ABB RobotStudio station: Lab5_RSSolution.rspag

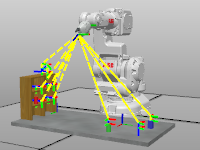
--- station ---
Station Lab5_RSSolution (saved by RobotStudio 20.4.9280.0)
Controller Lab5Controller
  mechanical unit ROB_1: IRB140_6_81_C_03, 6 joints, base frame (0, 0, 0) mm
Layout (positions relative to the parent item):
  - IRB140_6_81_C_03 [mechanism, from Robots\IRB140_6_81_C_G_03.rslib] at (0, 0, 0) mm; joint values [0, 0, 0, 0, 0.5236, 0] (rad or m)
  - HorizontalPlaneBoard [part]
  - WoodenRack [part]
  - PrismPiece [part] at (380, 400, 25) mm
  - CylinderPiece [part] at (580, 200, 25) mm, rotated rx 0 ry 0 rz -90 deg
  - HexagonalPrismPiece [part] at (502.54, -420.19, 127.78) mm, rotated rx 0 ry 0 rz -1.03 deg
  - Smart_Gripper_Servo_Fingers [mechanism, from Libraries\Smart_Gripper_Servo_Fingers.rslib] at (506.29, 0, 679.5) mm, rotated rx 180 ry 60 rz 180 deg; joint values [0.025] (rad or m)
  - PickAndPlaceLogic [smart component]
      signals: DI ActivateGripper, DI ReleaseGripper, DO PieceTaken
      connections:
        PickAndPlaceLogic.ActivateGripper -> Attacher.Execute
        PickAndPlaceLogic.ReleaseGripper -> Detacher.Execute
    - Attacher [smart component, from Components\Attacher.rslib]
        properties: Parent=Smart_Gripper_Servo_Fingers; Flange=0; Child=HexagonalPrismPiece; Mount=false; Offset=[0 0 0]; Orientation=[0 0 0]
    - Detacher [smart component, from Components\Detacher.rslib]
        properties: Child=HexagonalPrismPiece; KeepPosition=true
Attachment: Smart_Gripper_Servo_Fingers is attached to IRB140_6_81_C_03 / Link6
Station logic (signal -> signal, property => property):
  PickAndPlaceLogic.PieceTaken -> Lab5Controller.DI_01
  Lab5Controller.DO_02 -> PickAndPlaceLogic.ReleaseGripper
  Lab5Controller.DO_01 -> PickAndPlaceLogic.ActivateGripper

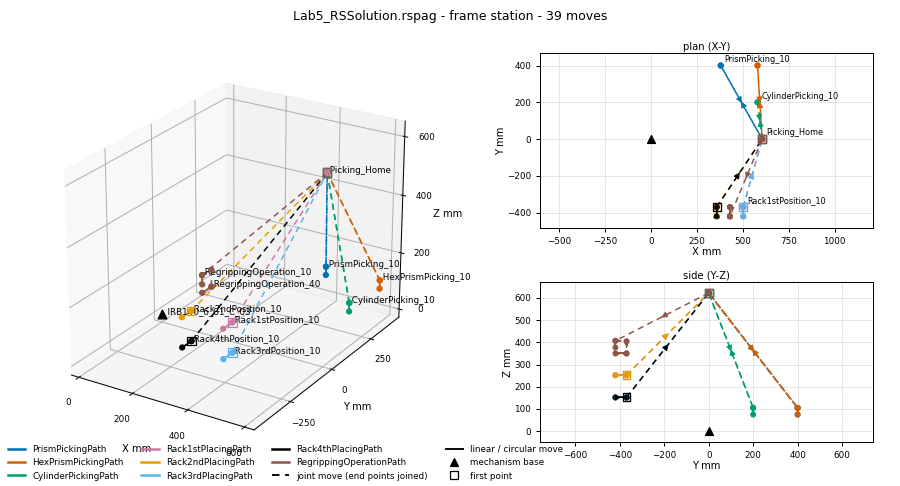
[picture p0: tool path of Lab5_RSSolution.rspag in frame station, 39 of 39 moves have a stored position in this frame; points joined in program order, loops and branches not executed]
--- Backups/Lab5Controller/RAPID/TASK1/PROGMOD/Module1.mod ---
MODULE Module1
        PERS tooldata Servo:=[TRUE,[[0,0,114.2],[1,0,0,0]],[0.215,[8.7,12.3,49.2],[1,0,0,0],0.00021,0.00024,0.00009]];
    TASK PERS wobjdata RackWorkObject:=[FALSE,TRUE,"",[[280,-400,25],[0.707107,0,0,-0.707107]],[[0,0,0],[1,0,0,0]]];
    TASK PERS wobjdata PiecesWorkObject:=[FALSE,TRUE,"",[[380,200,25],[1,0,0,0]],[[0,0,0],[1,0,0,0]]];
    CONST robtarget Picking_Home:=[[225.191752358,-200,597.4],[0.5,0,0.866025404,0],[0,0,0,0],[9E+09,9E+09,9E+09,9E+09,9E+09,9E+09]];
    CONST robtarget PrismPicking_10:=[[0,200,80],[0,0,1,0],[0,0,0,0],[9E+09,9E+09,9E+09,9E+09,9E+09,9E+09]];
    CONST robtarget PrismPicking_20:=[[0,200,50],[0,0,1,0],[0,0,0,0],[9E+09,9E+09,9E+09,9E+09,9E+09,9E+09]];
    CONST robtarget HexPrismPicking_10:=[[200,200,80],[0,0.258819045,0.965925826,0],[0,0,0,0],[9E+09,9E+09,9E+09,9E+09,9E+09,9E+09]];
    CONST robtarget HexPrismPicking_20:=[[200,200,50],[0,0.258819045,0.965925826,0],[0,0,0,0],[9E+09,9E+09,9E+09,9E+09,9E+09,9E+09]];
    CONST robtarget CylinderPicking_10:=[[200,0,80],[0,0.707106781,0.707106781,0],[0,0,1,0],[9E+09,9E+09,9E+09,9E+09,9E+09,9E+09]];
    CONST robtarget CylinderPicking_20:=[[200,0,50],[0,0.707106781,0.707106781,0],[0,0,0,0],[9E+09,9E+09,9E+09,9E+09,9E+09,9E+09]];
    CONST robtarget Rack1stPosition_10:=[[-30,222.5,227],[0.5,-0.5,0.5,-0.5],[-1,-2,0,0],[9E+09,9E+09,9E+09,9E+09,9E+09,9E+09]];
    CONST robtarget Rack1stPosition_20:=[[20,222.5,227],[0.5,-0.5,0.5,-0.5],[-1,-2,0,0],[9E+09,9E+09,9E+09,9E+09,9E+09,9E+09]];
    CONST robtarget Placing_Home:=[[-400,325.191800236,597.400057165],[0.353553394,-0.612372434,0.612372434,0.353553394],[0,0,0,0],[9E+09,9E+09,9E+09,9E+09,9E+09,9E+09]];
    CONST robtarget Rack2ndPosition_10:=[[-30,77.5,227],[0.5,-0.5,0.5,-0.5],[-1,-2,0,0],[9E+09,9E+09,9E+09,9E+09,9E+09,9E+09]];
    CONST robtarget Rack2ndPosition_20:=[[20,77.5,227],[0.5,-0.5,0.5,-0.5],[-1,-2,0,0],[9E+09,9E+09,9E+09,9E+09,9E+09,9E+09]];
    CONST robtarget Rack3rdPosition_10:=[[-30,222.5,127],[0.5,-0.5,0.5,-0.5],[-1,-2,0,0],[9E+09,9E+09,9E+09,9E+09,9E+09,9E+09]];
    CONST robtarget Rack3rdPosition_20:=[[20,222.5,127],[0.5,-0.5,0.5,-0.5],[-1,-2,0,0],[9E+09,9E+09,9E+09,9E+09,9E+09,9E+09]];
    CONST robtarget Rack4thPosition_10:=[[-30,77.5,127],[0.5,-0.5,0.5,-0.5],[-1,-2,0,0],[9E+09,9E+09,9E+09,9E+09,9E+09,9E+09]];
    CONST robtarget Rack4thPosition_20:=[[20,77.5,127],[0.5,-0.5,0.5,-0.5],[-1,-2,0,0],[9E+09,9E+09,9E+09,9E+09,9E+09,9E+09]];
    CONST robtarget RegrippingOperation_10:=[[20,150,382],[0,-0.707106781,0.707106781,0],[0,0,0,0],[9E+09,9E+09,9E+09,9E+09,9E+09,9E+09]];
    CONST robtarget RegrippingOperation_20:=[[20,150,352],[0,-0.707106781,0.707106781,0],[-1,0,-1,0],[9E+09,9E+09,9E+09,9E+09,9E+09,9E+09]];
    CONST robtarget RegrippingOperation_30:=[[-30,150,380],[0.27059805,-0.653281482,0.653281482,-0.27059805],[-1,-2,0,0],[9E+09,9E+09,9E+09,9E+09,9E+09,9E+09]];
    CONST robtarget RegrippingOperation_40:=[[-30,150,325],[0.5,-0.5,0.5,-0.5],[-1,-2,0,0],[9E+09,9E+09,9E+09,9E+09,9E+09,9E+09]];
    CONST robtarget RegrippingOperation_50:=[[20,150,325],[0.5,-0.5,0.5,-0.5],[-1,-2,0,0],[9E+09,9E+09,9E+09,9E+09,9E+09,9E+09]];


    PROC main()
        WaitDI DI_01, 1;
        HexPrismPickingPath;
        RegrippingOperationPath;
        Rack3rdPlacingPath;
    ENDPROC
    PROC PrismPickingPath()
        MoveJ Picking_Home,v200,z10,Servo\WObj:=PiecesWorkObject;
        MoveJ PrismPicking_10,v200,z10,Servo\WObj:=PiecesWorkObject;
        MoveL PrismPicking_20,v20,z1,Servo\WObj:=PiecesWorkObject;
        MoveL PrismPicking_10,v20,z1,Servo\WObj:=PiecesWorkObject;
        MoveJ Picking_Home,v200,z10,Servo\WObj:=PiecesWorkObject;
    ENDPROC
    PROC HexPrismPickingPath()
        MoveJ Picking_Home,v200,z10,Servo\WObj:=PiecesWorkObject;
        MoveJ HexPrismPicking_10,v200,z10,Servo\WObj:=PiecesWorkObject;
        MoveL HexPrismPicking_20,v20,z1,Servo\WObj:=PiecesWorkObject;
        setDO DO_01, 1;
        WaitTime 1;
        SetDO DO_01, 0;
        MoveL HexPrismPicking_10,v20,z1,Servo\WObj:=PiecesWorkObject;
        MoveJ Picking_Home,v200,z10,Servo\WObj:=PiecesWorkObject;
    ENDPROC
    PROC CylinderPickingPath()
        MoveJ Picking_Home,v200,z10,Servo\WObj:=PiecesWorkObject;
        MoveJ CylinderPicking_10,v200,z10,Servo\WObj:=PiecesWorkObject;
        MoveL CylinderPicking_20,v20,z1,Servo\WObj:=PiecesWorkObject;
        MoveL CylinderPicking_10,v20,z1,Servo\WObj:=PiecesWorkObject;
        MoveJ Picking_Home,v200,z10,Servo\WObj:=PiecesWorkObject;
    ENDPROC
    PROC Rack1stPlacingPath()
        MoveJ Rack1stPosition_10,v200,z10,Servo\WObj:=RackWorkObject;
        MoveL Rack1stPosition_20,v20,z1,Servo\WObj:=RackWorkObject;
        MoveL Rack1stPosition_10,v20,z1,Servo\WObj:=RackWorkObject;
        MoveJ Placing_Home,v200,z10,Servo\WObj:=RackWorkObject;
    ENDPROC
    PROC Rack2ndPlacingPath()
        MoveJ Rack2ndPosition_10,v200,z10,Servo\WObj:=RackWorkObject;
        MoveL Rack2ndPosition_20,v20,z1,Servo\WObj:=RackWorkObject;
        MoveL Rack2ndPosition_10,v20,z1,Servo\WObj:=RackWorkObject;
        MoveJ Placing_Home,v200,z10,Servo\WObj:=RackWorkObject;
    ENDPROC
    PROC Rack3rdPlacingPath()
        MoveJ Rack3rdPosition_10,v200,z10,Servo\WObj:=RackWorkObject;
        MoveL Rack3rdPosition_20,v20,z1,Servo\WObj:=RackWorkObject;
        SetDO DO_02, 1;
        WaitTime 1;
        SetDO DO_02, 0;
        MoveL Rack3rdPosition_10,v20,z1,Servo\WObj:=RackWorkObject;
        MoveJ Placing_Home,v200,z10,Servo\WObj:=RackWorkObject;
    ENDPROC
    PROC Rack4thPlacingPath()
        MoveJ Rack4thPosition_10,v200,z10,Servo\WObj:=RackWorkObject;
        MoveL Rack4thPosition_20,v20,z1,Servo\WObj:=RackWorkObject;
        MoveL Rack4thPosition_10,v20,z1,Servo\WObj:=RackWorkObject;
        MoveJ Placing_Home,v200,z10,Servo\WObj:=RackWorkObject;
    ENDPROC
    PROC RegrippingOperationPath()
        MoveJ Placing_Home,v200,z10,Servo\WObj:=RackWorkObject;
        MoveJ RegrippingOperation_10,v200,z10,Servo\WObj:=RackWorkObject;
        MoveL RegrippingOperation_20,v20,z1,Servo\WObj:=RackWorkObject;
        SetDO DO_02, 1;
        WaitTime 1;
        SetDO DO_02, 0;
        MoveL RegrippingOperation_10,v20,z1,Servo\WObj:=RackWorkObject;
        MoveJ RegrippingOperation_30,v200,z10,Servo\WObj:=RackWorkObject;
        MoveJ RegrippingOperation_40,v200,z10,Servo\WObj:=RackWorkObject;
        MoveL RegrippingOperation_50,v20,z1,Servo\WObj:=RackWorkObject;
        SetDO DO_01, 1;
        WaitTime 1;
        SetDO DO_01, 0;
        MoveL RegrippingOperation_40,v20,z1,Servo\WObj:=RackWorkObject;
    ENDPROC
ENDMODULE

--- Backups/Lab5Controller/RAPID/TASK1/SYSMOD/LINKEDM.sys ---
%%%
  VERSION:1
  LANGUAGE:ENGLISH
%%%

MODULE LINKEDM (SYSMODULE)

! FOLLOWER
!     Name of electronically linked follower axis used by operator at teach pendent.
      PERS string l_f_axis_name{5}       :=  ["",  "", "", "", ""];

!     Name of the mechanical unit for follower axis.
      PERS string l_f_mecunt_n{5}  :=  ["", "", "", "", ""];

!     Linked follower axis number in the mechanical unit (first axis in mech. unit is number 1).
      PERS num l_f_axis_no{5}      :=  [0,          0,   0,  0,  0];

! MASTER
!     Name of the mechanical unit for linked master axis.
      PERS string l_m_mecunt_n{5} :=  ["", "", "", "", ""];

!     Linked master axis number in the mechanical unit (first axis in mech. unit is number 1).
!     See axis number table in documentation for different master mechanical units.
      PERS num l_m_axis_no{5}     :=  [0,  0,  0,  0,  0];

! POSITION OFFSET
!     The increase of the allowed offset position between the master and follower
!     positions, used when starting AUTO mode. As soon as the offset is decreased
!     the old configurated parameter is used.
!     Example: 3 => the configurated value of allowed offset is increased 3 times.
      PERS num offset_ratio{5}       :=  [10,  10,   10,  10,  10];

! SPEED RATIO
!     Speed_ratio used in AUTO and JOG modes [ very_slow   slow    normal    fast]
!     Value 1 = max allowed manual speed.
      CONST num speed_ratio {20}      := [0.01, 0.01, 0.01, 0.01, 0.01,
                                          0.05, 0.05, 0.05, 0.05, 0.05,
                                          0.20, 0.20, 0.20, 0.20, 0.20,
                                          1.00, 1.00, 1.00, 1.00, 1.00];

! STEP SIZE
!     Displacement position used in JOG mode for each activation of positive or
!     negative movement.                  [very_short    short   normal   long]
!     Unit degees or meter.
      CONST num displacement {20}     := [0.001, 0.001, 0.001, 0.001, 0.001,
                                          0.005, 0.005, 0.005, 0.005, 0.005,
                                          0.020, 0.020, 0.020, 0.020, 0.020,
                                          0.100, 0.100, 0.100, 0.100, 0.100];


!-------------------------------------------------------------
 PROC Linked_m ()
      Linked_m_exe ;
 ENDPROC
ENDMODULE

--- Backups/Lab5Controller/SYSPAR/EIO.cfg ---
EIO:CFG_1.0:6:1::
#
EIO_SIGNAL:

      -Name "DI_01" -SignalType "DI" -Access "All"

      -Name "DI_02" -SignalType "DI" -Access "All"

      -Name "DI_03" -SignalType "DI" -Access "All"

      -Name "DO_01" -SignalType "DO" -Access "All"

      -Name "DO_02" -SignalType "DO"\
      -Label "Release the gripper fingers to home position" -Access "All"
